// TIA Portal V20 export
DATA_BLOCK "LPFE_AckAndResetBuffer"   // DB248
TITLE = Buffer of RequestOrderInfo messages
// Buffer to store Ack messages (1) until distributed
// stored: Access Published, MemoryReserve 100, Namespace PFE
   VAR
      buffer { ExternalAccessible := 'False'; ExternalVisible := 'False'; ExternalWritable := 'False'} : Array[0.._.LE_NUMBER_MESSAGES_ACK_BUFFER] of "LPFE_typePFEDataReqEnvelope";   // Buffer where ackmessages are taken from
      mgmtBuffer { ExternalAccessible := 'False'; ExternalVisible := 'False'; ExternalWritable := 'False'} : "LPFE_typeMsgBuffer";   // Mgmt Structure of buffer where ackmessages are taken from
   END_VAR
BEGIN
END_DATA_BLOCK
